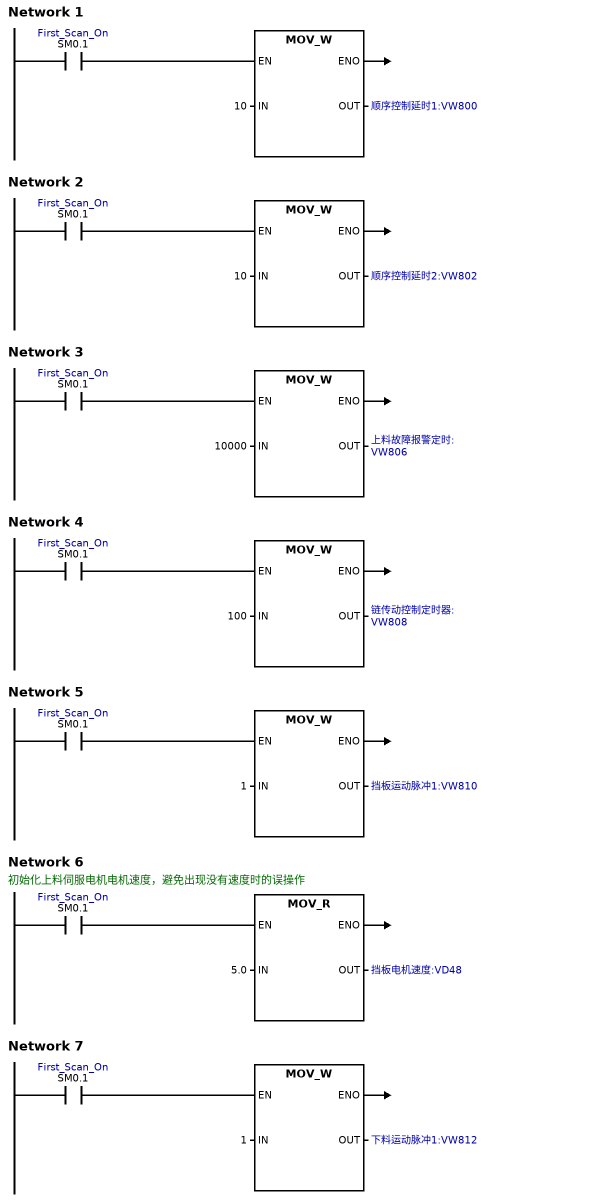
[picture p24: SBR20 networks 1-7]
Network 1
LD     First_Scan_On:SM0.1
MOVW   10, 顺序控制延时1:VW800
Network 2
LD     First_Scan_On:SM0.1
MOVW   10, 顺序控制延时2:VW802
Network 3
LD     First_Scan_On:SM0.1
MOVW   10000, 上料故障报警定时:VW806
Network 4
LD     First_Scan_On:SM0.1
MOVW   100, 链传动控制定时器:VW808
Network 5
LD     First_Scan_On:SM0.1
MOVW   1, 挡板运动脉冲1:VW810
Network 6
// 初始化上料伺服电机电机速度，避免出现没有速度时的误操作
LD     First_Scan_On:SM0.1
MOVR   5.0, 挡板电机速度:VD48
Network 7
LD     First_Scan_On:SM0.1
MOVW   1, 下料运动脉冲1:VW812
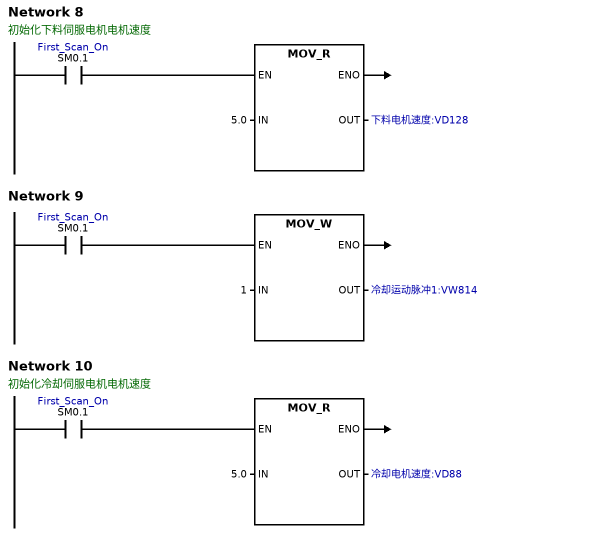
Network 8
// 初始化下料伺服电机电机速度
LD     First_Scan_On:SM0.1
MOVR   5.0, 下料电机速度:VD128
Network 9
LD     First_Scan_On:SM0.1
MOVW   1, 冷却运动脉冲1:VW814
Network 10
// 初始化冷却伺服电机电机速度
LD     First_Scan_On:SM0.1
MOVR   5.0, 冷却电机速度:VD88
END_SUBROUTINE_BLOCK
